					(* Valuto la posizione futura - Missione di Deposito *)
					IF (Mission^.YPick - IngombroOttimizzatoX_InPuntoDiDeposito/2 - OffsetSicurezza_Y <= WorkFootprint^[6].Y) OR //Posizione Pinza - Metà ingombro - Offset sicurezza <= Ingombro colonna 
						(Mission^.YPick + IngombroOttimizzatoX_InPuntoDiDeposito/2 + OffsetSicurezza_Y >= WorkFootprint^[5].Y) THEN //Posizione Pinza - Metà ingombro - Offset sicurezza <= Ingombro colonna 
							Pinza_InIngombroColonne_Destinazione := TRUE;
					ELSE
							Pinza_InIngombroColonne_Destinazione := FALSE;
					END_IF
					
					(* Valuto la posizione attuale Y e la posizione di destinazione Y e l'ingombro massimo che posso avere durante il transito *)
					IF (Mission^.YPick - IngombroOttimizzatoY_InTransito/2 - OffsetSicurezza_Y <= WorkFootprint^[6].Y) OR //Posizione Pinza - Metà ingombro - Offset sicurezza <= Ingombro colonna 
						(Mission^.YPick + IngombroOttimizzatoY_InTransito/2 + OffsetSicurezza_Y >= WorkFootprint^[5].Y) THEN //Posizione Pinza - Metà ingombro - Offset sicurezza <= Ingombro colonna 
							Pinza_InIngombroColonne_Transito := TRUE;
					ELSE
							Pinza_InIngombroColonne_Transito := FALSE;
					END_IF
						
				PALLETTIZZATORE_SX: // Colonna 6:SX, 5:DX
					(* Valuto la posizione attuale *)
					IF (ModuleAX_Y^.Ax^.Status.ActPosition - IngombroY/2 - OffsetSicurezza_Y <= WorkFootprint^[5].Y) OR //Posizione Pinza - Metà ingombro - Offset sicurezza <= Ingombro colonna 
						(ModuleAX_Y^.Ax^.Status.ActPosition + IngombroY/2 + OffsetSicurezza_Y >= WorkFootprint^[6].Y) THEN //Posizione Pinza - Metà ingombro - Offset sicurezza <= Ingombro colonna 
							Pinza_InIngombroColonne_Attuale := TRUE;
					ELSE
							Pinza_InIngombroColonne_Attuale := FALSE;
					END_IF
					(* Valuto la posizione futura - Missione di prelievo *)
					IF (Mission^.YPick - IngombroOttimizzatoX_InPuntoDiPrelievo/2 - OffsetSicurezza_Y <= WorkFootprint^[5].Y) OR //Posizione Pinza - Metà ingombro - Offset sicurezza <= Ingombro colonna 
						(Mission^.YPick + IngombroOttimizzatoX_InPuntoDiPrelievo/2 + OffsetSicurezza_Y >= WorkFootprint^[6].Y) THEN //Posizione Pinza - Metà ingombro - Offset sicurezza <= Ingombro colonna 
							Pinza_InIngombroColonne_Destinazione := TRUE;
					ELSE
							Pinza_InIngombroColonne_Destinazione := FALSE;
					END_IF
					
					(* Valuto la posizione futura - Missione di Deposito *)
					IF (Mission^.YPick - IngombroOttimizzatoX_InPuntoDiDeposito/2 - OffsetSicurezza_Y <= WorkFootprint^[5].Y) OR //Posizione Pinza - Metà ingombro - Offset sicurezza <= Ingombro colonna 
						(Mission^.YPick + IngombroOttimizzatoX_InPuntoDiDeposito/2 + OffsetSicurezza_Y >= WorkFootprint^[6].Y) THEN //Posizione Pinza - Metà ingombro - Offset sicurezza <= Ingombro colonna 
							Pinza_InIngombroColonne_Destinazione := TRUE;
					ELSE
							Pinza_InIngombroColonne_Destinazione := FALSE;
					END_IF
					
					(* Valuto la posizione attuale Y e la posizione di destinazione Y e l'ingombro massimo che posso avere durante il transito *)
					IF (Mission^.YPick - IngombroOttimizzatoY_InTransito/2 - OffsetSicurezza_Y <= WorkFootprint^[5].Y) OR //Posizione Pinza - Metà ingombro - Offset sicurezza <= Ingombro colonna 
						(Mission^.YPick + IngombroOttimizzatoY_InTransito/2 + OffsetSicurezza_Y >= WorkFootprint^[6].Y) THEN //Posizione Pinza - Metà ingombro - Offset sicurezza <= Ingombro colonna 
							Pinza_InIngombroColonne_Transito := TRUE;
					ELSE
							Pinza_InIngombroColonne_Transito := FALSE;
					END_IF
			END_CASE		
			(* Se sono in ingombro nella posizione attuale o nella posizione di destinazione, devo andare fuori-ingombro con la Y *)
			IF (Pinza_InIngombroColonne_Attuale OR Pinza_InIngombroColonne_Destinazione OR Pinza_InIngombroColonne_Transito) THEN 
				IF (AsseXInFinestraDiRiposo AND AsseYInFinestraDiRiposo AND AsseJInFinestraDiRiposo) THEN //Se sono in finestra di riposo con tutti gli assi non devo andare fuori-ingombro con la Y
					FuoriIngombroYNecessarioTMP := FALSE;
				ELSE
					FuoriIngombroYNecessarioTMP := TRUE;
				END_IF
			ELSE
				FuoriIngombroYNecessarioTMP := FALSE;
			END_IF
		END_IF
	WAMANAGER_CICLO_PRELIEVO_PACCO_END:
		CalcolaIngombro := TRUE;	
		
	WAMANAGER_CICLO_DEPOSITO_PACCO_RUN:
	
		IF CalcolaIngombro THEN
			CalcolaIngombro := FALSE;
			(* Definisco il tipo di area in cui si trova a lavorare il pallettizzatore *)
			AreaInLavoroPositiva := FALSE;
			AreaInLavoroNegativa := FALSE;
			AreaInLavoroPositivaNegativa := FALSE; 
			
			IF ModuleAx_X^.Ax^.AxRef^.NcToPlc.ActPos >= (WorkFootprint^[5].X + WorkFootprint^[5].XDim) AND 	//se la piazzola di prelievo ha quota maggiore rispetto le colonne centrali
				WorkArea^[Mission^.PPlace].X >= (WorkFootprint^[5].X + WorkFootprint^[5].XDim)  THEN //la piazzola di deposito è nella campata positiva
					AreaInLavoroPositiva := TRUE;
			ELSIF ModuleAx_X^.Ax^.AxRef^.NcToPlc.ActPos <= WorkFootprint^[5].X AND 	//se la piazzola di prelievo ha quota maggiore della piazzola di deposito e
				WorkArea^[Mission^.PPlace].X <= WorkFootprint^[5].X  THEN //la piazzola di deposito è nella campata negativa
					AreaInLavoroNegativa := TRUE;
			ELSE
				AreaInLavoroPositiva := FALSE;
				AreaInLavoroNegativa := FALSE;
				AreaInLavoroPositivaNegativa := TRUE;
			END_IF
			
			(**************************************************************************************************************************************************)
			(* Ingombro ottimizzato della pinza sul punto di prelievo *)
			(**************************************************************************************************************************************************)
			IngombroOttimizzatoX_InPuntoDiPrelievo := ABS(IngombroSuperficialePinzaMAX * SIN(deg_to_rad((ATAN(Larghezza/Lunghezza)*1/0.017+ Mission^.JPick))));
			IngombroOttimizzatoY_InPuntoDiPrelievo := ABS(IngombroSuperficialePinzaMAX * COS(deg_to_rad((ATAN(Larghezza/Lunghezza)*1/0.017+ Mission^.JPick))));
			(**************************************************************************************************************************************************)
			(* Ingombro ottimizzato della pinza sul punto di deposito *)
			(**************************************************************************************************************************************************)
			IngombroOttimizzatoX_InPuntoDiDeposito := ABS(IngombroSuperficialePinzaMAX * SIN(deg_to_rad((ATAN(Larghezza/Lunghezza)*1/0.017+ Mission^.JPlace))));
			IngombroOttimizzatoY_InPuntoDiDeposito := ABS(IngombroSuperficialePinzaMAX * COS(deg_to_rad((ATAN(Larghezza/Lunghezza)*1/0.017+ Mission^.JPlace))));
						
			(**************************************************************************************************************************************************)
			(**************************************************************************************************************************************************)
						
			(* Valuto la direzione della X *)
			DirezioneXPositiva := TFDirezioneAssePositiva(Posizione_Attuale:=ModuleAX_X^.Ax^.Status.ActPosition,Posizione_Finale:=Mission^.XPick);
			DirezioneXNegativa := NOT DirezioneXPositiva;
				
			(* Valuto se gli assi sono in finestra di prelievo *)
			AsseXInFinestraDiRiposo := TFAsseInFinestra(Posizione_Attuale:=ModuleAx_X^.Ax^.AxRef^.NcToPlc.ActPos,Posizione_Finale:=Mission^.XPick,FinestraDiControllo:=10);
			AsseYInFinestraDiRiposo := TFAsseInFinestra(Posizione_Attuale:=ModuleAx_Y^.Ax^.AxRef^.NcToPlc.ActPos,Posizione_Finale:=Mission^.YPick,FinestraDiControllo:=10);
			AsseJInFinestraDiRiposo := TFAsseInFinestra(Posizione_Attuale:=ModuleAx_J^.Ax^.AxRef^.NcToPlc.ActPos,Posizione_Finale:=Mission^.JPick,FinestraDiControllo:=5);
			(* Valuto se gli assi sono in finestra di destinazione *)
			AsseXInFinestraDiDestinazione := TFAsseInFinestra(Posizione_Attuale:=ModuleAx_X^.Ax^.AxRef^.NcToPlc.ActPos,Posizione_Finale:=Mission^.XPick,FinestraDiControllo:=10);
			AsseYInFinestraDiDestinazione := TFAsseInFinestra(Posizione_Attuale:=ModuleAx_Y^.Ax^.AxRef^.NcToPlc.ActPos,Posizione_Finale:=Mission^.YPick,FinestraDiControllo:=10);
			AsseJInFinestraDiDestinazione := TFAsseInFinestra(Posizione_Attuale:=ModuleAx_J^.Ax^.AxRef^.NcToPlc.ActPos,Posizione_Finale:=Mission^.JPick,FinestraDiControllo:=5);
			
			(**************************************************************************************************************************************************)
			(* Ingombro MASSIMO della pinza durante il transito *)
			(**************************************************************************************************************************************************)
			//Calcolo ingombro attuale
			IngombroOttimizzatoX_InTransito := ABS(IngombroSuperficialePinzaMAX * SIN(deg_to_rad((ATAN(Larghezza/Lunghezza)*1/0.017+ ModuleAx_J^.Ax^.AxRef^.NcToPlc.ActPos)))); //Ingombro Attuale direzione X
			IngombroOttimizzatoY_InTransito := ABS(IngombroSuperficialePinzaMAX * COS(deg_to_rad((ATAN(Larghezza/Lunghezza)*1/0.017+ ModuleAx_J^.Ax^.AxRef^.NcToPlc.ActPos)))); //Ingombro Attuale direzione Y		
			IF NOT AsseJInFinestraDiDestinazione THEN
				IF REAL_TO_INT(ModuleAx_J^.Ax^.AxRef^.NcToPlc.ActPos) <= REAL_TO_INT(Mission^.JPick) THEN
					FOR Angolo := REAL_TO_INT(ModuleAx_J^.Ax^.AxRef^.NcToPlc.ActPos) TO REAL_TO_INT(Mission^.JPick)  DO
						IF IngombroOttimizzatoX_InTransito < ABS(IngombroSuperficialePinzaMAX * SIN(deg_to_rad((ATAN(Larghezza/Lunghezza)*1/0.017+ Angolo)))) THEN
							IngombroOttimizzatoX_InTransito := ABS(IngombroSuperficialePinzaMAX * SIN(deg_to_rad((ATAN(Larghezza/Lunghezza)*1/0.017+ Angolo)))) ;
						END_IF
						IF IngombroOttimizzatoY_InTransito < ABS(IngombroSuperficialePinzaMAX * COS(deg_to_rad((ATAN(Larghezza/Lunghezza)*1/0.017+ Angolo)))) THEN
							IngombroOttimizzatoY_InTransito := ABS(IngombroSuperficialePinzaMAX * COS(deg_to_rad((ATAN(Larghezza/Lunghezza)*1/0.017+ Angolo))));
						END_IF
					END_FOR
				END_IF
			END_IF
		
			(* Valutazione colonne in base al verso del pallettizzatore *)
			CASE VERSO_PALLETTIZZATORE OF
				PALLETTIZZATORE_DX:	// Colonna 6:DX, 5:SX
					(* Valuto la posizione attuale *)
					IF (ModuleAX_Y^.Ax^.Status.ActPosition - IngombroY/2 - OffsetSicurezza_Y <= WorkFootprint^[6].Y) OR //Posizione Pinza - Metà ingombro - Offset sicurezza <= Ingombro colonna 
						(ModuleAX_Y^.Ax^.Status.ActPosition + IngombroY/2 + OffsetSicurezza_Y >= WorkFootprint^[5].Y) THEN //Posizione Pinza - Metà ingombro - Offset sicurezza <= Ingombro colonna 
							Pinza_InIngombroColonne_Attuale := TRUE;
					ELSE
							Pinza_InIngombroColonne_Attuale := FALSE;
					END_IF
					(* Valuto la posizione futura - Missione di prelievo *)
					IF (Mission^.YPick - IngombroOttimizzatoX_InPuntoDiPrelievo/2 - OffsetSicurezza_Y <= WorkFootprint^[6].Y) OR //Posizione Pinza - Metà ingombro - Offset sicurezza <= Ingombro colonna 
						(Mission^.YPick + IngombroOttimizzatoX_InPuntoDiPrelievo/2 + OffsetSicurezza_Y >= WorkFootprint^[5].Y) THEN //Posizione Pinza - Metà ingombro - Offset sicurezza <= Ingombro colonna 
							Pinza_InIngombroColonne_Destinazione := TRUE;
					ELSE
							Pinza_InIngombroColonne_Destinazione := FALSE;
					END_IF
					
					(* Valuto la posizione futura - Missione di Deposito *)
					IF (Mission^.YPick - IngombroOttimizzatoX_InPuntoDiDeposito/2 - OffsetSicurezza_Y <= WorkFootprint^[6].Y) OR //Posizione Pinza - Metà ingombro - Offset sicurezza <= Ingombro colonna 
						(Mission^.YPick + IngombroOttimizzatoX_InPuntoDiDeposito/2 + OffsetSicurezza_Y >= WorkFootprint^[5].Y) THEN //Posizione Pinza - Metà ingombro - Offset sicurezza <= Ingombro colonna 
							Pinza_InIngombroColonne_Destinazione := TRUE;
					ELSE
							Pinza_InIngombroColonne_Destinazione := FALSE;
					END_IF
					
					(* Valuto la posizione attuale Y e la posizione di destinazione Y e l'ingombro massimo che posso avere durante il transito *)
					IF (Mission^.YPick - IngombroOttimizzatoY_InTransito/2 - OffsetSicurezza_Y <= WorkFootprint^[6].Y) OR //Posizione Pinza - Metà ingombro - Offset sicurezza <= Ingombro colonna 
						(Mission^.YPick + IngombroOttimizzatoY_InTransito/2 + OffsetSicurezza_Y >= WorkFootprint^[5].Y) THEN //Posizione Pinza - Metà ingombro - Offset sicurezza <= Ingombro colonna 
							Pinza_InIngombroColonne_Transito := TRUE;
					ELSE
							Pinza_InIngombroColonne_Transito := FALSE;
					END_IF
						
				PALLETTIZZATORE_SX: // Colonna 6:SX, 5:DX
					(* Valuto la posizione attuale *)
					IF (ModuleAX_Y^.Ax^.Status.ActPosition - IngombroY/2 - OffsetSicurezza_Y <= WorkFootprint^[5].Y) OR //Posizione Pinza - Metà ingombro - Offset sicurezza <= Ingombro colonna 
						(ModuleAX_Y^.Ax^.Status.ActPosition + IngombroY/2 + OffsetSicurezza_Y >= WorkFootprint^[6].Y) THEN //Posizione Pinza - Metà ingombro - Offset sicurezza <= Ingombro colonna 
							Pinza_InIngombroColonne_Attuale := TRUE;
					ELSE
							Pinza_InIngombroColonne_Attuale := FALSE;
					END_IF
					(* Valuto la posizione futura - Missione di prelievo *)
					IF (Mission^.YPick - IngombroOttimizzatoX_InPuntoDiPrelievo/2 - OffsetSicurezza_Y <= WorkFootprint^[5].Y) OR //Posizione Pinza - Metà ingombro - Offset sicurezza <= Ingombro colonna 
						(Mission^.YPick + IngombroOttimizzatoX_InPuntoDiPrelievo/2 + OffsetSicurezza_Y >= WorkFootprint^[6].Y) THEN //Posizione Pinza - Metà ingombro - Offset sicurezza <= Ingombro colonna 
							Pinza_InIngombroColonne_Destinazione := TRUE;
					ELSE
							Pinza_InIngombroColonne_Destinazione := FALSE;
					END_IF
					
					(* Valuto la posizione futura - Missione di Deposito *)
					IF (Mission^.YPick - IngombroOttimizzatoX_InPuntoDiDeposito/2 - OffsetSicurezza_Y <= WorkFootprint^[5].Y) OR //Posizione Pinza - Metà ingombro - Offset sicurezza <= Ingombro colonna 
						(Mission^.YPick + IngombroOttimizzatoX_InPuntoDiDeposito/2 + OffsetSicurezza_Y >= WorkFootprint^[6].Y) THEN //Posizione Pinza - Metà ingombro - Offset sicurezza <= Ingombro colonna 
							Pinza_InIngombroColonne_Destinazione := TRUE;
					ELSE
							Pinza_InIngombroColonne_Destinazione := FALSE;
					END_IF
					
					(* Valuto la posizione attuale Y e la posizione di destinazione Y e l'ingombro massimo che posso avere durante il transito *)
					IF (Mission^.YPick - IngombroOttimizzatoY_InTransito/2 - OffsetSicurezza_Y <= WorkFootprint^[5].Y) OR //Posizione Pinza - Metà ingombro - Offset sicurezza <= Ingombro colonna 
						(Mission^.YPick + IngombroOttimizzatoY_InTransito/2 + OffsetSicurezza_Y >= WorkFootprint^[6].Y) THEN //Posizione Pinza - Metà ingombro - Offset sicurezza <= Ingombro colonna 
							Pinza_InIngombroColonne_Transito := TRUE;
					ELSE
							Pinza_InIngombroColonne_Transito := FALSE;
					END_IF
			END_CASE		
			(* Se sono in ingombro nella posizione attuale o nella posizione di destinazione, devo andare fuori-ingombro con la Y *)
			IF (Pinza_InIngombroColonne_Attuale OR Pinza_InIngombroColonne_Destinazione OR Pinza_InIngombroColonne_Transito) THEN 
				IF (AsseXInFinestraDiRiposo AND AsseYInFinestraDiRiposo AND AsseJInFinestraDiRiposo) THEN //Se sono in finestra di riposo con tutti gli assi non devo andare fuori-ingombro con la Y
					FuoriIngombroYNecessarioTMP := FALSE;
				ELSE
					FuoriIngombroYNecessarioTMP := TRUE;
				END_IF
			ELSE
				FuoriIngombroYNecessarioTMP := FALSE;
			END_IF
		END_IF
		
	WAMANAGER_CICLO_DEPOSITO_PACCO_END:
		CalcolaIngombro := TRUE;	
	
END_CASE

TFCalcoliFuoriIngombriColonne := TRUE;

END_FUNCTION

(* stored: Version 1.1.0.1, ProductVersion 3.1.4024.11
   POU TFCalcoliFuoriIngombriColonne_old: Id {b12b0920-5560-445f-9c3e-c3d670b7b1b7}, SpecialFunc None *)
